{attribute 'linkalways'} 
{attribute 'no_explicit_call' := 'This FB is a CLASS and must be accessed using methods or properties'}
{attribute 'enable_dynamic_creation'}
FUNCTION_BLOCK FINAL AND_LWORD EXTENDS Node
VAR
	in1 : _LWORD(0);
	in2 : _LWORD(0);
	out : _LWORD(0);
END_VAR

METHOD PUBLIC Clone : I_Node
VAR
	pNode : POINTER TO AND_LWORD;
END_VAR
pNode := __NEW(AND_LWORD);
Clone := pNode^;
END_METHOD

METHOD FB_init : BOOL
VAR_INPUT
	bInitRetains : BOOL; // if TRUE, the retain variables are initialized (warm start / cold start)
	bInCopyCode : BOOL;  // if TRUE, the instance afterwards gets moved into the copy code (online change)
END_VAR
AddInput('in1',THIS^.in1);
AddInput('in2',THIS^.in2);
AddOutput('out', THIS^.out);
END_METHOD

METHOD PROTECTED OnExecute
VAR
END_VAR
out.Value := in1.Value AND in2.Value;
END_METHOD

END_FUNCTION_BLOCK

(* stored: Version 1.1.0.1, ProductVersion 3.1.4024.15
   POU AND_LWORD: Id {e879bed0-0d92-4dd6-9bd2-6ba55f44aee1}, SpecialFunc None
   Folder Constructor: Id {eeaac217-6d27-4cb4-8a76-8c83e401ab42}
   Method Clone: Id {0c299b0c-45c0-4552-a8e6-01a70acda42c}
   Method FB_init: Id {15b4df93-f5a8-4c8a-b21a-7db4a01ce4cc}
   Method OnExecute: Id {55d268bf-8ba1-47bf-abcc-fb39b96fff32} *)
